// TIA Portal project "Level station" (V15)

(* hardware
DEVICE "S71500/ET200MP station_1"  S7-1500 station
   slot 0: "Rail_0"  Rack  6ES7 590-1***0-0AA0
   slot 1: "Level_control"  CPU 1512C-1 PN  6ES7 512-1CK01-0AB0  V2.5
      slot 3: "CPU display_1"  6ES7591-1AA00-0AA0
DEVICE "S71500/ET200MP station_2"  S7-1500 station
   slot 0: "Rail_0"  Rack  6ES7 590-1***0-0AA0
   slot 1: "Flow_control"  CPU 1512C-1 PN  6ES7 512-1CK01-0AB0  V2.5
      slot 3: "CPU display_1"  6ES7591-1AA00-0AA0
*)

// ===== PLC "Level_control"  CPU 1512C-1 PN =====

VAR_GLOBAL   // PLC tag table "Default tag table"
   "Tag_1" AT %M0.0 : Bool;
   "Tag_2" AT %IW272 : Word;
   "Tag_3" AT %MD3 : Real;
   "Tag_4" AT %MD7 : Real;
   "Tag_5" AT %QW290 : Int;
   "Tag_6" AT %M0.1 : Bool;
   "Tag_7" AT %M0.2 : Bool;
   "Tag_8" AT %MD11 : DWord;
   "Tag_10" AT %QW0 : Int;
   "Tag_11" AT %IW0 : Int;
   "Tag_9" AT %MD50 : Real;
   "Tag_12" AT %M0.6 : Bool;
END_VAR

DATA_BLOCK "Data_block_1"   // DB1
{ S7_Optimized_Access := 'FALSE' }
VERSION : 0.1
   VAR
      K_c : Real;
      tau_i : Real;
      tau_d : Real;
      Mk : Real;
      "Mk-1" : Real := 0.0;
      ek : Real;
      "ek-1" : Real;
      "ek-2" : Real;
      delta_t : Real := 0.25;
   END_VAR
BEGIN
END_DATA_BLOCK

FUNCTION "Block_1" : Void   // FC1, LAD
{ S7_Optimized_Access := 'TRUE' }
VERSION : 0.1
   VAR_INPUT
      In : Int;
      PIWmin : Real;
      PIWmax : Real;
      x_max : Real;
      x_min : Real;
   END_VAR
   VAR_OUTPUT
      Out : Real;
   END_VAR
   VAR_TEMP
      Temp1 : DInt;
      Temp2 : Real;
      Temp3 : Real;
      Temp4 : Real;
      Temp5 : Real;
      Temp6 : Real;
      Temp7 : Real;
   END_VAR
BEGIN

REGION Network 1
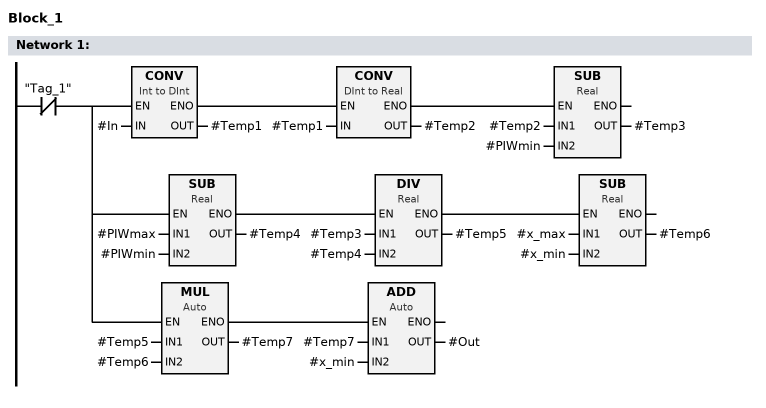
   RUNG wire#powerrail
      I_Contact( "Tag_1" )
      wire#w1
      { S7_Templates := "[SrcType := Int, DestType := DInt]" } Convert(in := #In, out => #Temp1)
      { S7_Templates := "[SrcType := DInt, DestType := Real]" } Convert(in := #Temp1, out => #Temp2)
      { S7_Templates := "SrcType := Real" } Sub(in1 := #Temp2, in2 := #PIWmin, out => #Temp3)
   END_RUNG
   RUNG wire#w1
      { S7_Templates := "SrcType := Real" } Sub(in1 := #PIWmax, in2 := #PIWmin, out => #Temp4)
      { S7_Templates := "SrcType := Real" } Div(in1 := #Temp3, in2 := #Temp4, out => #Temp5)
      { S7_Templates := "SrcType := Real" } Sub(in1 := #x_max, in2 := #x_min, out => #Temp6)
   END_RUNG
   RUNG wire#w1
      Mul(in1 := #Temp5, in2 := #Temp6, out => #Temp7)
      Add(in1 := #Temp7, in2 := #x_min, out => #Out)
   END_RUNG
   // the same network as SCL:
   IF NOT "Tag_1" THEN
       #Temp1 := INT_TO_DINT(#In);
       #Temp2 := DINT_TO_REAL(#Temp1);
       #Temp3 := #Temp2 - #PIWmin;
       #Temp4 := #PIWmax - #PIWmin;
       #Temp5 := #Temp3 / #Temp4;
       #Temp6 := #x_max - #x_min;
       #Temp7 := #Temp5 * #Temp6;
       #Out := #Temp7 + #x_min;
   END_IF;
END_REGION
END_FUNCTION

FUNCTION "Block_2" : Void   // FC2, LAD
{ S7_Optimized_Access := 'TRUE' }
VERSION : 0.1
   VAR_INPUT
      mv : Real;
      u_max : Real;
      u_min : Real;
      PQWmax : Real;
      PQWmin : Real;
   END_VAR
   VAR_OUTPUT
      PQWx : Int;
   END_VAR
   VAR_TEMP
      Temp3 : Real;
      Temp4 : Real;
      Temp5 : Real;
      Temp6 : Real;
      Temp7 : Real;
      Temp8 : Real;
      Temp9 : DInt;
   END_VAR
BEGIN

REGION Network 1
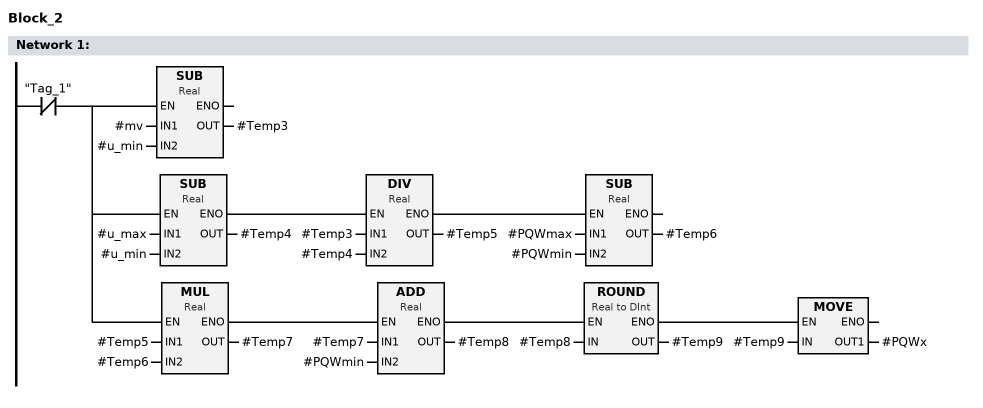
   RUNG wire#powerrail
      I_Contact( "Tag_1" )
      wire#w1
      { S7_Templates := "SrcType := Real" } Sub(in1 := #mv, in2 := #u_min, out => #Temp3)
   END_RUNG
   RUNG wire#w1
      { S7_Templates := "SrcType := Real" } Sub(in1 := #u_max, in2 := #u_min, out => #Temp4)
      { S7_Templates := "SrcType := Real" } Div(in1 := #Temp3, in2 := #Temp4, out => #Temp5)
      { S7_Templates := "SrcType := Real" } Sub(in1 := #PQWmax, in2 := #PQWmin, out => #Temp6)
   END_RUNG
   RUNG wire#w1
      { S7_Templates := "SrcType := Real" } Mul(in1 := #Temp5, in2 := #Temp6, out => #Temp7)
      { S7_Templates := "SrcType := Real" } Add(in1 := #Temp7, in2 := #PQWmin, out => #Temp8)
      { S7_Templates := "[SrcType := Real, DestType := DInt]" } Round(in := #Temp8, out => #Temp9)
      Move(in := #Temp9, out1 => #PQWx)
   END_RUNG
   // the same network as SCL:
   IF NOT "Tag_1" THEN
       #Temp3 := #mv - #u_min;
       #Temp4 := #u_max - #u_min;
       #Temp5 := #Temp3 / #Temp4;
       #Temp6 := #PQWmax - #PQWmin;
       #Temp7 := #Temp5 * #Temp6;
       #Temp8 := #Temp7 + #PQWmin;
       #Temp9 := ROUND(#Temp8);
       #PQWx := #Temp9;
   END_IF;
END_REGION
END_FUNCTION

FUNCTION "Block_3" : Void   // FC3, LAD
{ S7_Optimized_Access := 'TRUE' }
VERSION : 0.1
   VAR_INPUT
      K_c : Real;
      tau_i : Real;
      tau_d : Real;
      delta_t : Real;
      ek : Real;
      "ek-1" : Real;
      "ek-2" : Real;
      "MVk-1" : Real;
   END_VAR
   VAR_OUTPUT
      MVk : Real;
   END_VAR
   VAR_TEMP
      temp1 : Real;
      temp2 : Real;
      temp3 : Real;
      temp4 : Real;
      temp5 : Real;
      temp6 : Real;
      temp7 : Real;
      temp8 : Real;
      temp9 : Real;
      temp10 : Real;
      temp11 : Real;
      temp12 : Real;
      temp13 : Real;
      temp14 : Real;
      temp15 : Real;
   END_VAR
BEGIN

REGION Network 1
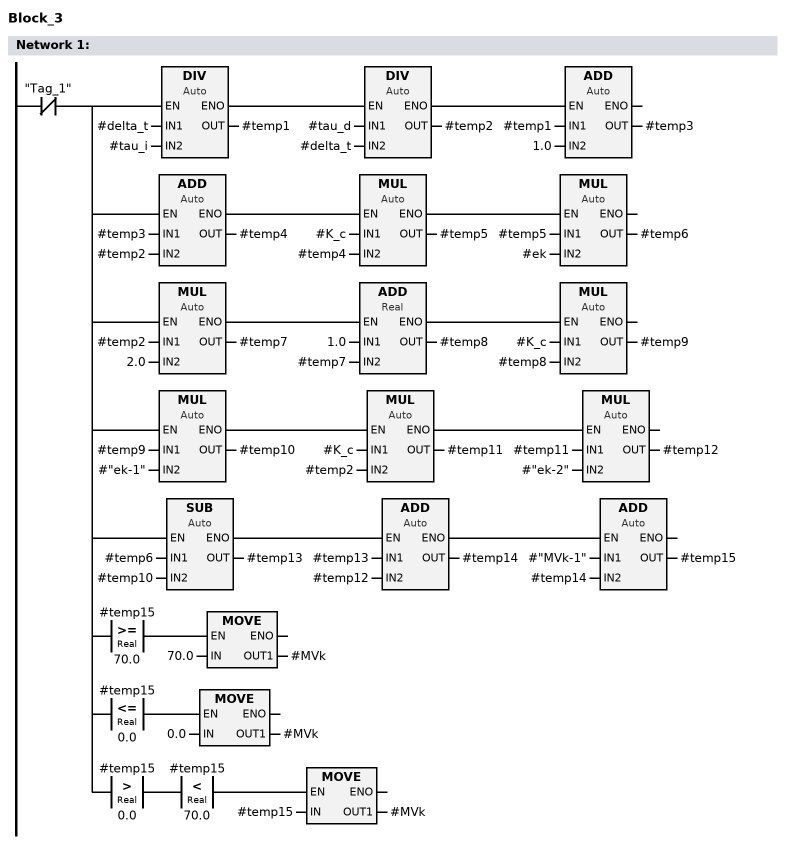
   RUNG wire#powerrail
      I_Contact( "Tag_1" )
      wire#w1
      Div(in1 := #delta_t, in2 := #tau_i, out => #temp1)
      Div(in1 := #tau_d, in2 := #delta_t, out => #temp2)
      Add(in1 := #temp1, in2 := 1.0, out => #temp3)
   END_RUNG
   RUNG wire#w1
      Add(in1 := #temp3, in2 := #temp2, out => #temp4)
      Mul(in1 := #K_c, in2 := #temp4, out => #temp5)
      Mul(in1 := #temp5, in2 := #ek, out => #temp6)
   END_RUNG
   RUNG wire#w1
      Mul(in1 := #temp2, in2 := 2.0, out => #temp7)
      { S7_Templates := "SrcType := Real" } Add(in1 := 1.0, in2 := #temp7, out => #temp8)
      Mul(in1 := #K_c, in2 := #temp8, out => #temp9)
   END_RUNG
   RUNG wire#w1
      Mul(in1 := #temp9, in2 := #"ek-1", out => #temp10)
      Mul(in1 := #K_c, in2 := #temp2, out => #temp11)
      Mul(in1 := #temp11, in2 := #"ek-2", out => #temp12)
   END_RUNG
   RUNG wire#w1
      Sub(in1 := #temp6, in2 := #temp10, out => #temp13)
      Add(in1 := #temp13, in2 := #temp12, out => #temp14)
      Add(in1 := #"MVk-1", in2 := #temp14, out => #temp15)
   END_RUNG
   RUNG wire#w1
      { S7_Templates := "SrcType := Real" } GE_Contact(in1 := #temp15, in2 := 70.0)
      Move(in := 70.0, out1 => #MVk)
   END_RUNG
   RUNG wire#w1
      { S7_Templates := "SrcType := Real" } LE_Contact(in1 := #temp15, in2 := 0.0)
      Move(in := 0.0, out1 => #MVk)
   END_RUNG
   RUNG wire#w1
      { S7_Templates := "SrcType := Real" } GT_Contact(in1 := #temp15, in2 := 0.0)
      { S7_Templates := "SrcType := Real" } LT_Contact(in1 := #temp15, in2 := 70.0)
      Move(in := #temp15, out1 => #MVk)
   END_RUNG
   // the same network as SCL:
   IF NOT "Tag_1" THEN
       #temp1 := #delta_t / #tau_i;
       #temp2 := #tau_d / #delta_t;
       #temp3 := #temp1 + 1.0;
       #temp4 := #temp3 + #temp2;
       #temp5 := #K_c * #temp4;
       #temp6 := #temp5 * #ek;
       #temp7 := #temp2 * 2.0;
       #temp8 := 1.0 + #temp7;
       #temp9 := #K_c * #temp8;
       #temp10 := #temp9 * #"ek-1";
       #temp11 := #K_c * #temp2;
       #temp12 := #temp11 * #"ek-2";
       #temp13 := #temp6 - #temp10;
       #temp14 := #temp13 + #temp12;
       #temp15 := #"MVk-1" + #temp14;
   END_IF;
   IF NOT "Tag_1" AND (#temp15 >= 70.0) THEN #MVk := 70.0; END_IF;
   IF NOT "Tag_1" AND (#temp15 <= 0.0) THEN #MVk := 0.0; END_IF;
   IF NOT "Tag_1" AND (#temp15 > 0.0) AND (#temp15 < 70.0) THEN #MVk := #temp15; END_IF;
END_REGION
END_FUNCTION

FUNCTION "PI" : Void   // FC4, LAD
{ S7_Optimized_Access := 'TRUE' }
VERSION : 0.1
   VAR_INPUT
      K_c : Real;
      tau_i : Real;
      delta_t : Real;
      ek : Real;
      "ek-1" : Real;
      "ek-2" : Real;
      "MVk-1" : Real;
   END_VAR
   VAR_OUTPUT
      MVk : Real;
   END_VAR
   VAR_TEMP
      temp1 : Real;
      temp2 : Real;
      temp3 : Real;
      temp4 : Real;
      temp5 : Real;
      temp6 : Real;
      temp7 : Real;
      temp8 : Real;
      temp9 : Real;
      temp10 : Real;
      temp11 : Real;
      temp12 : Real;
      temp13 : Real;
      temp14 : Real;
      temp15 : Real;
   END_VAR
BEGIN

REGION Network 1
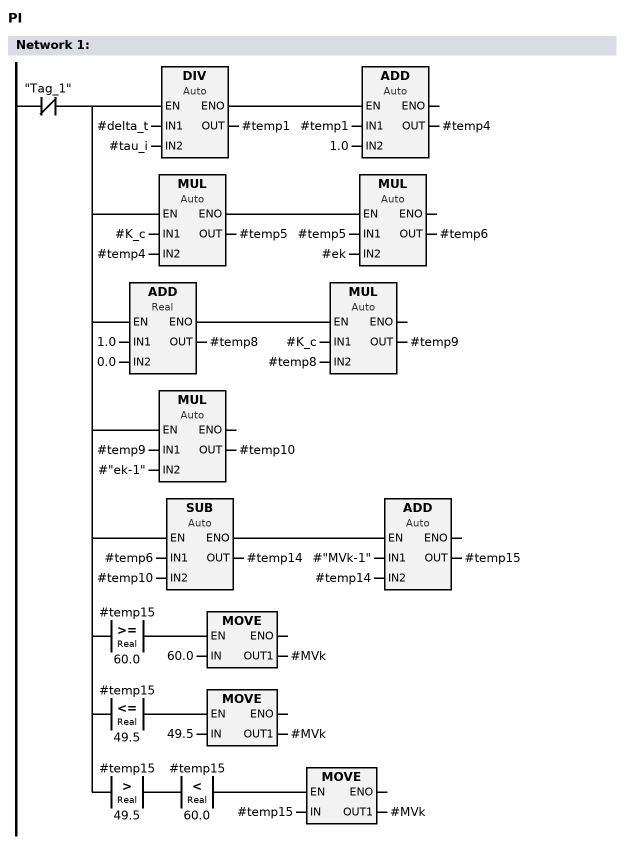
   RUNG wire#powerrail
      I_Contact( "Tag_1" )
      wire#w1
      Div(in1 := #delta_t, in2 := #tau_i, out => #temp1)
      Add(in1 := #temp1, in2 := 1.0, out => #temp4)
   END_RUNG
   RUNG wire#w1
      Mul(in1 := #K_c, in2 := #temp4, out => #temp5)
      Mul(in1 := #temp5, in2 := #ek, out => #temp6)
   END_RUNG
   RUNG wire#w1
      { S7_Templates := "SrcType := Real" } Add(in1 := 1.0, in2 := 0.0, out => #temp8)
      Mul(in1 := #K_c, in2 := #temp8, out => #temp9)
   END_RUNG
   RUNG wire#w1
      Mul(in1 := #temp9, in2 := #"ek-1", out => #temp10)
   END_RUNG
   RUNG wire#w1
      Sub(in1 := #temp6, in2 := #temp10, out => #temp14)
      Add(in1 := #"MVk-1", in2 := #temp14, out => #temp15)
   END_RUNG
   RUNG wire#w1
      { S7_Templates := "SrcType := Real" } GE_Contact(in1 := #temp15, in2 := 60.0)
      Move(in := 60.0, out1 => #MVk)
   END_RUNG
   RUNG wire#w1
      { S7_Templates := "SrcType := Real" } LE_Contact(in1 := #temp15, in2 := 49.5)
      Move(in := 49.5, out1 => #MVk)
   END_RUNG
   RUNG wire#w1
      { S7_Templates := "SrcType := Real" } GT_Contact(in1 := #temp15, in2 := 49.5)
      { S7_Templates := "SrcType := Real" } LT_Contact(in1 := #temp15, in2 := 60.0)
      Move(in := #temp15, out1 => #MVk)
   END_RUNG
   // the same network as SCL:
   IF NOT "Tag_1" THEN
       #temp1 := #delta_t / #tau_i;
       #temp4 := #temp1 + 1.0;
       #temp5 := #K_c * #temp4;
       #temp6 := #temp5 * #ek;
       #temp8 := 1.0 + 0.0;
       #temp9 := #K_c * #temp8;
       #temp10 := #temp9 * #"ek-1";
       #temp14 := #temp6 - #temp10;
       #temp15 := #"MVk-1" + #temp14;
   END_IF;
   IF NOT "Tag_1" AND (#temp15 >= 60.0) THEN #MVk := 60.0; END_IF;
   IF NOT "Tag_1" AND (#temp15 <= 49.5) THEN #MVk := 49.5; END_IF;
   IF NOT "Tag_1" AND (#temp15 > 49.5) AND (#temp15 < 60.0) THEN #MVk := #temp15; END_IF;
END_REGION
END_FUNCTION

FUNCTION "P" : Void   // FC5, LAD
{ S7_Optimized_Access := 'TRUE' }
VERSION : 0.1
   VAR_INPUT
      K_c : Real;
      MVk_1 : Real;
      ek : Real;
   END_VAR
   VAR_OUTPUT
      MVk : Real;
   END_VAR
   VAR_TEMP
      temp3 : Real;
      temp2 : Real;
      temp1 : Real;
   END_VAR
BEGIN

REGION Network 1
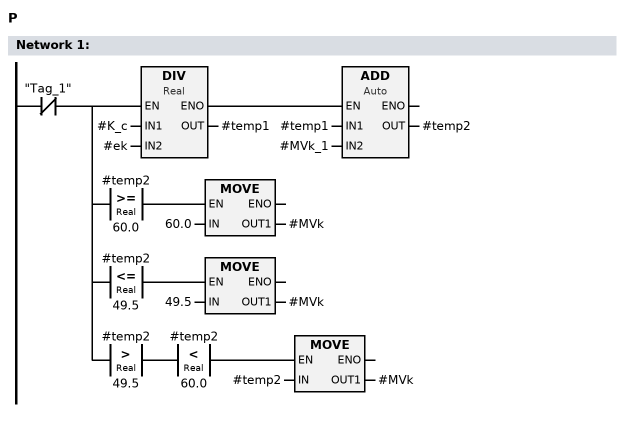
   RUNG wire#powerrail
      I_Contact( "Tag_1" )
      wire#w1
      { S7_Templates := "SrcType := Real" } Div(in1 := #K_c, in2 := #ek, out => #temp1)
      Add(in1 := #temp1, in2 := #MVk_1, out => #temp2)
   END_RUNG
   RUNG wire#w1
      { S7_Templates := "SrcType := Real" } GE_Contact(in1 := #temp2, in2 := 60.0)
      Move(in := 60.0, out1 => #MVk)
   END_RUNG
   RUNG wire#w1
      { S7_Templates := "SrcType := Real" } LE_Contact(in1 := #temp2, in2 := 49.5)
      Move(in := 49.5, out1 => #MVk)
   END_RUNG
   RUNG wire#w1
      { S7_Templates := "SrcType := Real" } GT_Contact(in1 := #temp2, in2 := 49.5)
      { S7_Templates := "SrcType := Real" } LT_Contact(in1 := #temp2, in2 := 60.0)
      Move(in := #temp2, out1 => #MVk)
   END_RUNG
   // the same network as SCL:
   IF NOT "Tag_1" THEN
       #temp1 := #K_c / #ek;
       #temp2 := #temp1 + #MVk_1;
   END_IF;
   IF NOT "Tag_1" AND (#temp2 >= 60.0) THEN #MVk := 60.0; END_IF;
   IF NOT "Tag_1" AND (#temp2 <= 49.5) THEN #MVk := 49.5; END_IF;
   IF NOT "Tag_1" AND (#temp2 > 49.5) AND (#temp2 < 60.0) THEN #MVk := #temp2; END_IF;
END_REGION
END_FUNCTION

ORGANIZATION_BLOCK "Main"   // OB1, LAD, ProgramCycle
TITLE = "Main Program Sweep (Cycle)"
{ S7_Optimized_Access := 'FALSE' }
VERSION : 0.1
   VAR_TEMP
      EV_CLASS : Byte;   // Bits 0-3 = 1:Coming event, Bits 4-7 = 1:Event class 1
      SCAN_1 : Byte;   // 1:Initial call of the OB, 3: Call 2-n of the OB
      PRIORITY : Byte;   // Priority of OB Execution
      OB_NUMBR : Byte;   // OB number
      RESERVED_1 : Byte;   // Reserved for system
      RESERVED_2 : Byte;   // Reserved for system
      PREV_CYCLE : Int;   // Previous program cycle time (milliseconds)
      MIN_CYCLE : Int;   // Minimum program cycle time (milliseconds)
      MAX_CYCLE : Int;   // Maximum program cycle time (milliseconds)
      DATE_TIME : Date_And_Time;   // Date and time OB started
      OB1_EV_CLASS : Byte;
      OB1_SCAN_1 : Byte;
   END_VAR
   VAR_TEMP   // added for the SCL form of the ladder/FBD networks
      _w1 : Bool;
   END_VAR
BEGIN

REGION Network 1
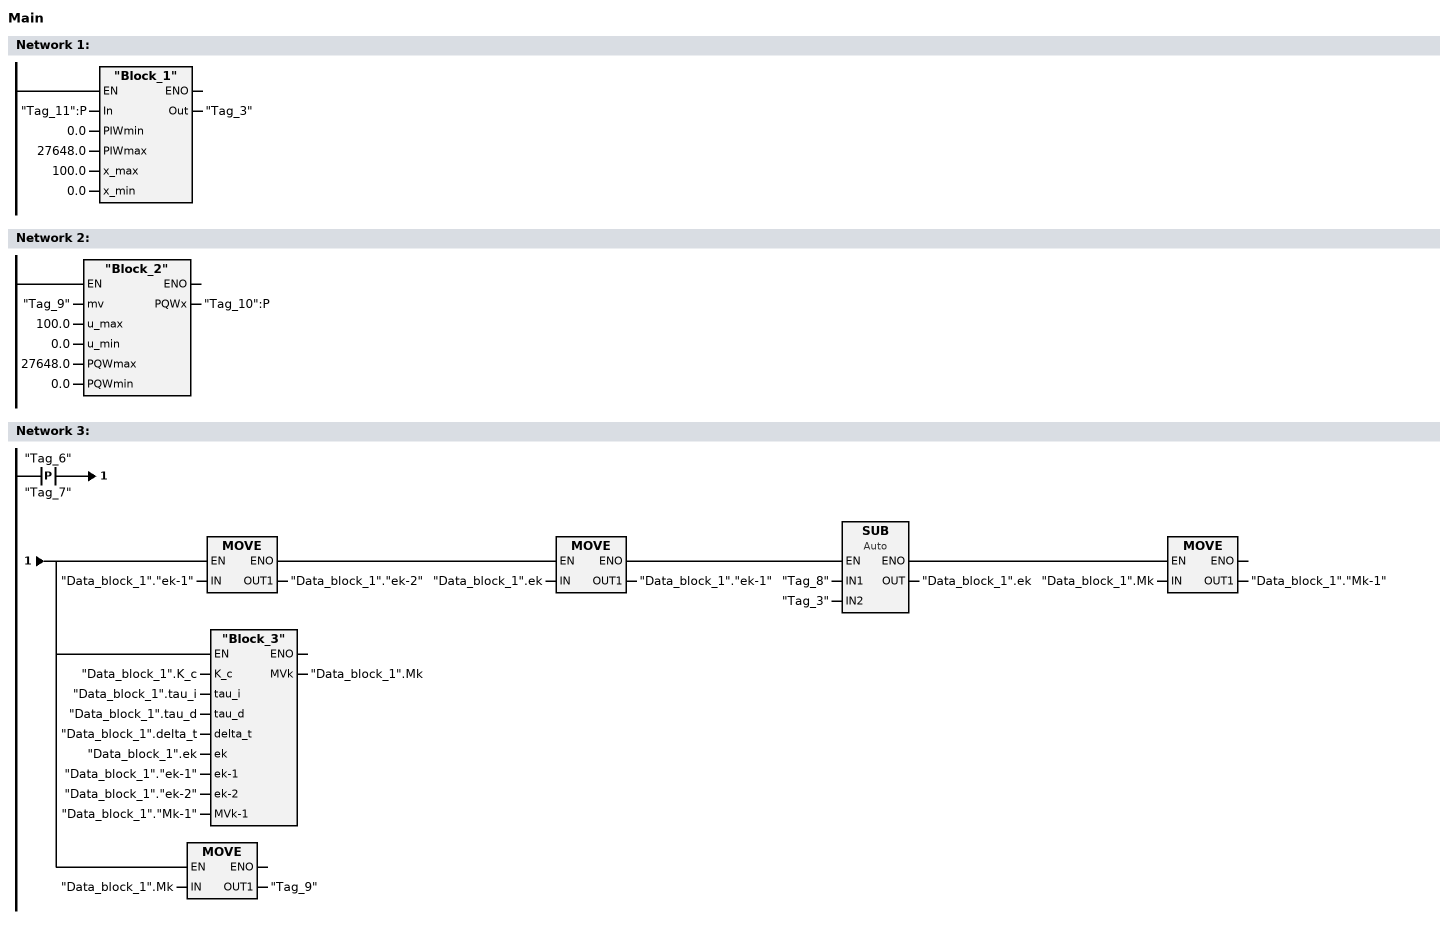
   RUNG wire#powerrail
      "Block_1"(In := "Tag_11":P, PIWmin := 0.0, PIWmax := 27648.0, x_max := 100.0, x_min := 0.0, Out => "Tag_3")
   END_RUNG
   // the same network as SCL:
   "Block_1"(In := "Tag_11":P, PIWmin := 0.0, PIWmax := 27648.0, x_max := 100.0, x_min := 0.0, Out => "Tag_3");
END_REGION

REGION Network 2
   RUNG wire#powerrail
      "Block_2"(mv := "Tag_9", u_max := 100.0, u_min := 0.0, PQWmax := 27648.0, PQWmin := 0.0, PQWx => "Tag_10":P)
   END_RUNG
   // the same network as SCL:
   "Block_2"(mv := "Tag_9", u_max := 100.0, u_min := 0.0, PQWmax := 27648.0, PQWmin := 0.0, PQWx => "Tag_10":P);
END_REGION

REGION Network 3
   RUNG wire#powerrail
      P_Contact(operand := "Tag_6", bit := "Tag_7")
      wire#w1
      Move(in := "Data_block_1"."ek-1", out1 => "Data_block_1"."ek-2")
      Move(in := "Data_block_1".ek, out1 => "Data_block_1"."ek-1")
      Sub(in1 := "Tag_8", in2 := "Tag_3", out => "Data_block_1".ek)
      Move(in := "Data_block_1".Mk, out1 => "Data_block_1"."Mk-1")
   END_RUNG
   RUNG wire#w1
      "Block_3"(K_c := "Data_block_1".K_c, tau_i := "Data_block_1".tau_i, tau_d := "Data_block_1".tau_d, delta_t := "Data_block_1".delta_t, ek := "Data_block_1".ek, "ek-1" := "Data_block_1"."ek-1", "ek-2" := "Data_block_1"."ek-2", "MVk-1" := "Data_block_1"."Mk-1", MVk => "Data_block_1".Mk)
   END_RUNG
   RUNG wire#w1
      Move(in := "Data_block_1".Mk, out1 => "Tag_9")
   END_RUNG
   // the same network as SCL:
   #_w1 := "Tag_6" AND NOT "Tag_7";   // rising edge of "Tag_6"
   "Tag_7" := "Tag_6";
   IF #_w1 THEN
       "Data_block_1"."ek-2" := "Data_block_1"."ek-1";
       "Data_block_1"."ek-1" := "Data_block_1".ek;
       "Data_block_1".ek := "Tag_8" - "Tag_3";
       "Data_block_1"."Mk-1" := "Data_block_1".Mk;
       "Block_3"(K_c := "Data_block_1".K_c,
                 tau_i := "Data_block_1".tau_i,
                 tau_d := "Data_block_1".tau_d,
                 delta_t := "Data_block_1".delta_t,
                 ek := "Data_block_1".ek,
                 "ek-1" := "Data_block_1"."ek-1",
                 "ek-2" := "Data_block_1"."ek-2",
                 "MVk-1" := "Data_block_1"."Mk-1",
                 MVk => "Data_block_1".Mk);
       "Tag_9" := "Data_block_1".Mk;
   END_IF;
END_REGION
END_ORGANIZATION_BLOCK

ORGANIZATION_BLOCK "Cyclic interrupt"   // OB35, LAD, CyclicInterrupt
{ S7_Optimized_Access := 'TRUE' }
VERSION : 0.1
   VAR_INPUT
      Initial_Call : Bool;   // Initial call of this OB
      Event_Count : Int;   // Events discarded
   END_VAR
BEGIN

REGION Network 1
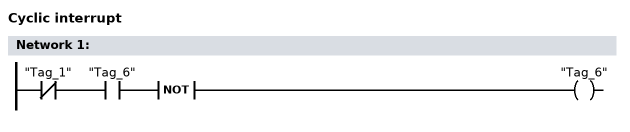
   RUNG wire#powerrail
      I_Contact( "Tag_1" )
      Contact( "Tag_6" )
      Not()
      Coil( "Tag_6" )
   END_RUNG
   // the same network as SCL:
   "Tag_6" := NOT (NOT "Tag_1" AND "Tag_6");
END_REGION
END_ORGANIZATION_BLOCK

// ===== PLC "Flow_control"  CPU 1512C-1 PN =====

ORGANIZATION_BLOCK "Main"   // OB1, LAD, ProgramCycle
TITLE = "Main Program Sweep (Cycle)"
{ S7_Optimized_Access := 'TRUE' }
VERSION : 0.1
   VAR_INPUT
      Initial_Call : Bool;   // Initial call of this OB
      Remanence : Bool;   // =True, if remanent data are available
   END_VAR
BEGIN
END_ORGANIZATION_BLOCK